(* IEC 61131-3 sources: Concurso_PLC/plc/codesys/03_FUN, 5 files *)

(* ---- FC_ColorFromSensors.st ---- *)
(* Convierte las dos senales digitales de vision en un color.
   S6.1 (Green Raw Material) -> GREEN    S6.2 (Blue Raw Material) -> BLUE
   Ninguna, o ambas a la vez (lectura incoherente) -> NONE *)
FUNCTION FC_ColorFromSensors : E_Color
VAR_INPUT
    xGreen : BOOL;   (* S6.1 *)
    xBlue  : BOOL;   (* S6.2 *)
END_VAR

IF xGreen AND NOT xBlue THEN
    FC_ColorFromSensors := E_Color.GREEN;
ELSIF xBlue AND NOT xGreen THEN
    FC_ColorFromSensors := E_Color.BLUE;
ELSE
    FC_ColorFromSensors := E_Color.NONE;
END_IF

(* ---- FC_FifoClear.st ---- *)
FUNCTION FC_FifoClear : BOOL
VAR_IN_OUT
    stFifo : ST_Fifo;
END_VAR

stFifo.iHead  := 0;
stFifo.iCount := 0;
FC_FifoClear  := TRUE;

(* ---- FC_FifoPack.st ---- *)
(* Empaqueta los colores de la cola en una WORD para el HMI:
   2 bits por pieza (01 = verde, 10 = azul), la primera pieza de la cola en los bits 0-1.
   Muestra como maximo 8 piezas. *)
FUNCTION FC_FifoPack : WORD
VAR_IN_OUT
    stFifo : ST_Fifo;
END_VAR
VAR
    k      : INT;
    iIdx   : INT;
    wPack  : WORD;
END_VAR

wPack := 0;
FOR k := 0 TO MIN(stFifo.iCount, 8) - 1 DO
    iIdx  := (stFifo.iHead + k) MOD GVL_Param.FIFO_SIZE;
    wPack := wPack OR SHL(INT_TO_WORD(TO_INT(stFifo.aItem[iIdx])), 2 * k);
END_FOR
FC_FifoPack := wPack;

(* ---- FC_FifoPop.st ---- *)
(* Extrae el primer color de la cola. Devuelve NONE si esta vacia. *)
FUNCTION FC_FifoPop : E_Color
VAR_IN_OUT
    stFifo : ST_Fifo;
END_VAR

IF stFifo.iCount <= 0 THEN
    FC_FifoPop := E_Color.NONE;
ELSE
    FC_FifoPop := stFifo.aItem[stFifo.iHead];
    stFifo.iHead := (stFifo.iHead + 1) MOD GVL_Param.FIFO_SIZE;
    stFifo.iCount := stFifo.iCount - 1;
END_IF

(* ---- FC_FifoPush.st ---- *)
(* Inserta un color al final de la cola. Devuelve FALSE si la cola esta llena. *)
FUNCTION FC_FifoPush : BOOL
VAR_IN_OUT
    stFifo : ST_Fifo;
END_VAR
VAR_INPUT
    eItem  : E_Color;
END_VAR
VAR
    iTail  : INT;
END_VAR

IF stFifo.iCount >= GVL_Param.FIFO_SIZE THEN
    FC_FifoPush := FALSE;
ELSE
    iTail := (stFifo.iHead + stFifo.iCount) MOD GVL_Param.FIFO_SIZE;
    stFifo.aItem[iTail] := eItem;
    stFifo.iCount := stFifo.iCount + 1;
    FC_FifoPush := TRUE;
END_IF
